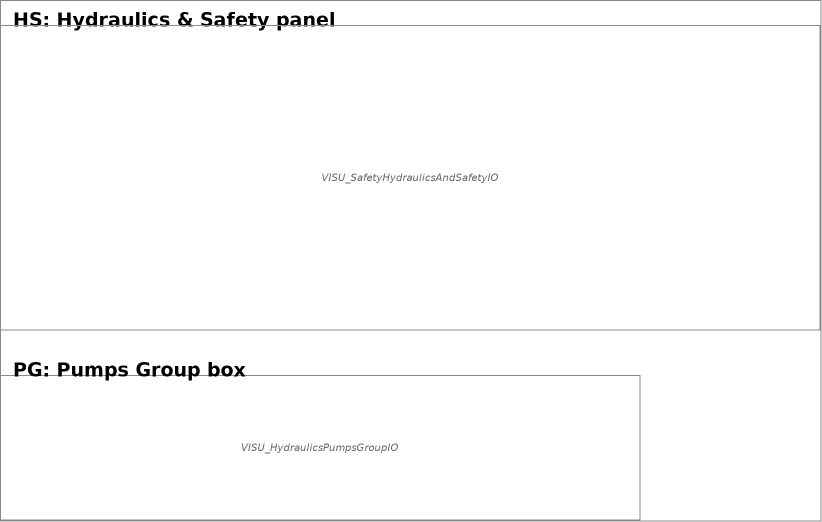
VISUALIZATION VISU_HydraulicsIO  // 822x522
VAR_IN_OUT
	ref : HydraulicsIO;
    ref_safetyIO : SafetyIO;
    widget : HydraulicsIOWidget;
END_VAR
    Label (10,5 350x30), "HS: Hydraulics & Safety panel"
    Frame (0,25 820x305)
        shows VISU_SafetyHydraulicsAndSafetyIO(ref := ref_safetyIO.parts.hydraulicsAndSafety, widget := widget.hydraulicsAndSafety)
        shows VISU_SafetyDomeAccessIO()
    Frame (0,375 640x145)
        shows VISU_HydraulicsPumpsGroupIO(ref := ref.parts.pumpsGroup, widget := widget.pumpsGroup)
        shows VISU_SafetyDomeAccessIO()
    Label (10,355 350x30), "PG: Pumps Group box"
END_VISUALIZATION

(* stored: Version 1.1.0.1, ProductVersion 3.1.4019.2
   Visu VISU_HydraulicsIO: Id {33cd705c-992d-46c7-a15b-ed88bba8adc8} *)
